// TIA Portal V19 export
VAR_GLOBAL   // PLC tag table "Standard_IO"
   I_LeftSensorPaperRem_42B1 AT %I100.0 : Bool;   // Left sensor paper remover   {ExternalAccessible false}
   I_RightSensorPaperRem_42B2 AT %I100.1 : Bool;   // Right sensor paper remover   {ExternalAccessible false}
   I_EmptySensorPaperMag_40B1 AT %I100.2 : Bool;   // Magazine – Empty sensor   {ExternalAccessible false}
   I_ColorSensor1PaperMag_40B2 AT %I100.3 : Bool;   // Magazine – Colour sensor 1   {ExternalAccessible false}
   I_ColorSensor2PaperMag_40B3 AT %I100.4 : Bool;   // Magazine – Colour sensor 2   {ExternalAccessible false}
   I_ColorSensor3PaperMag_40B4 AT %I100.5 : Bool;   // Magazine – Colour sensor 3   {ExternalAccessible false}
   I_GimbalLockedFerrobotics AT %I101.0 : Bool;   // AOK – Gimbal locked   {ExternalAccessible false}
   I_PositionOkExcentricFerrobotics AT %I101.1 : Bool;   // AOK – Excentric position Ok   {ExternalAccessible false}
   I_GreaseSensorX AT %I102.0 : Bool;   // Robot X axis - Grease pressure sensor   {ExternalAccessible false}
   I_GreaseSensorZ AT %I102.2 : Bool;   // Robot Z axis - Grease pressure sensor   {ExternalAccessible false}
   I_YAxisLoadSecured_48B1 AT %I102.4 : Bool;   // Robot Z axis - Load secured   {ExternalAccessible false}
   I_YAxisClampingInactive_48B2 AT %I102.5 : Bool;   // Robot Z axis - Clamping Inactive   {ExternalAccessible false}
   IW_DistanceSensor_42B4 AT %IW600 : Int;   // Robot - distance sensor   {ExternalAccessible false}
   O_SignalToweGreenLight AT %Q100.0 : Bool;   // Light towers - green light   {ExternalAccessible false}
   O_SignalToweOrangeLight AT %Q100.1 : Bool;   // Light towers - orange light   {ExternalAccessible false}
   O_SignalToweRedLight AT %Q100.2 : Bool;   // Light towers - red light   {ExternalAccessible false}
   O_SignalToweHorn AT %Q100.3 : Bool;   // Light towers - horn   {ExternalAccessible false}
   OST_SendRobot AT %Q104.0 : "stSendRobot";   //    {ExternalAccessible false}
   IST_RecieveRobot AT %I104.0 : "stRecieveRobot";   //    {ExternalAccessible false}
   OST_SendMaster AT %Q181.0 : "stSlaveToMaster";   //    {ExternalAccessible false}
   IST_RecieveMaster AT %I181.0 : "stMasterToSlave";   //    {ExternalAccessible false}
   O_UnlockExcentricGear1 AT %Q169.0 : Bool;   // Enable valve to unlock excentric Gear 1   {ExternalAccessible false}
   O_UnlockExcentricGear2 AT %Q169.1 : Bool;   // Enable valve to unlock excentric Gear 2   {ExternalAccessible false}
   O_UnlockExcentricGear3 AT %Q169.2 : Bool;   // Enable valve to unlock excentric Gear 3   {ExternalAccessible false}
   O_LockGimball AT %Q169.3 : Bool;   // Enable valve to lock Gimball   {ExternalAccessible false}
   OW_SetForceTarget AT %QW173 : Word;   //    {ExternalAccessible false}
   OW_SetForceZero AT %QW175 : Word;   //    {ExternalAccessible false}
   OB_SetTimeRamp AT %QB177 : Byte;   //    {ExternalAccessible false}
   OW_SetSpeed AT %QW178 : Word;   //    {ExternalAccessible false}
   IW_ActForce AT %IW173 : Word;   //    {ExternalAccessible false}
   IW_ActPosition AT %IW175 : Word;   //    {ExternalAccessible false}
   IB_ActContactState AT %IB177 : Byte;   //    {ExternalAccessible false}
   IW_ActErrorCode AT %IW178 : Word;   //    {ExternalAccessible false}
   O_EnablePumpX AT %Q101.0 : Bool;   // Robot X axis - Enable grease pump   {ExternalAccessible false}
   O_EnablePumpZ AT %Q101.1 : Bool;   // Robot Z axis - Enable grease pump   {ExternalAccessible false}
   I_PinionSensorX AT %I90.0 : Bool;   // Robot X axis - Sensor detection rotation pinion   {ExternalAccessible false}
   I_PinionSensorZ AT %I90.1 : Bool;   // Robot Z axis - Sensor detection rotation pinion   {ExternalAccessible false}
   O_BlowingSensor AT %Q100.7 : Bool;   // Blow FerRobotic sensor on remove disk station   {ExternalAccessible false}
   O_CloseVacuumValve AT %Q100.6 : Bool;   // Close Vacuum valve during disk changing   {ExternalAccessible false}
   I_VacuumValveClosed AT %I101.6 : Bool;   // Vacuum valve closed   {ExternalAccessible false}
   I_VacuumValveOpen AT %I101.7 : Bool;   // Vacuum valve open   {ExternalAccessible false}
   IB_Inout100 AT %IB100 : Byte;   //    {ExternalAccessible false}
   IB_Inout101 AT %IB101 : Byte;   //    {ExternalAccessible false}
   IB_Inout102 AT %IB102 : Byte;   //    {ExternalAccessible false}
   IB_Inout103 AT %IB103 : Byte;   //    {ExternalAccessible false}
   IB_Fast90 AT %IB90 : Byte;   //    {ExternalAccessible false}
   OB_Output100 AT %QB100 : Byte;   //    {ExternalAccessible false}
   OB_Output101 AT %QB101 : Byte;   //    {ExternalAccessible false}
   IW_Input602 AT %IW602 : Int;   // Robot - distance sensor   {ExternalAccessible false}
   IW_Input604 AT %IW604 : Int;   //    {ExternalAccessible false}
   IW_Input606 AT %IW606 : Int;   //    {ExternalAccessible false}
   I_FeedbackPowerFerRobotic AT %I507.0 : Bool;   // Feedback from safety relay for 24V safety power of FerRobotic Head   {ExternalAccessible false}
   I_FeedbackRevPowerFerRobotic AT %I507.1 : Bool;   // Feedback Reverse from safety relay for 24V safety power of FerRobotic Head   {ExternalAccessible false}
END_VAR
